TYPE
    ST_MotorCommand :
    STRUCT
        Forward  : BOOL;
        Backward : BOOL;
        Stopped  : BOOL;
    END_STRUCT
END_TYPE

(* stored: Version 1.1.0.1, ProductVersion 3.1.4024.13
   DUT ST_MotorCommand: Id {9006aa1e-5fb8-4b24-910d-fa6538e7d06f} *)
